FUNCTION_BLOCK Sensor_Sense
VAR_INPUT
	mxEnable: BOOL;
END_VAR
VAR_OUTPUT
	Product:STRING;
	mxINVALIDPRODUCT:BOOL;
	mxREDPLATE:BOOL;
	mxYELLOWPLATE:BOOL;
	mxBLUEPLATE:BOOL;
	mxREDCYLINDER:BOOL;
	mxYELLOWCYLINDER:BOOL;
	mxBLUECYLINDER:BOOL;
	mxREDOCTAGON:BOOL;
	mxYELLOWOCTAGON:BOOL;
	mxBLUEOCTAGON:BOOL;
	mxREDCONTAINER:BOOL;
	mxYELLOWCONTAINER:BOOL;
	mxBLUECONTAINER:BOOL;
END_VAR
VAR
	Sensor_Sense:BYTE;
END_VAR

IF mxEnable THEN
	Sensor_Sense.1:=gvl.ixInductiveSensor1;
	Sensor_Sense.2:=gvl.ixInductiveSensor2;
	Sensor_Sense.3:=gvl.ixInductiveSensor3;
	Sensor_Sense.4:=gvl.ixInductiveSensor4;
END_IF

IF Sensor_Sense = 0 OR Sensor_Sense = 4 OR Sensor_Sense = 2 OR Sensor_Sense = 6 THEN
 	Product:='InvalidPart';
	mxINVALIDPRODUCT:=FALSE;
END_IF

IF Sensor_Sense=16 THEN
	Product:='Blue Container';
	mxREDPLATE:=FALSE;
	mxYELLOWPLATE:=FALSE;
	mxBLUEPLATE:=FALSE;
	mxREDCYLINDER:=FALSE;
	mxYELLOWCYLINDER:=FALSE;
	mxBLUECYLINDER:=FALSE;
	mxREDOCTAGON:=FALSE;
	mxYELLOWOCTAGON:=FALSE;
	mxBLUEOCTAGON:=FALSE;
	mxREDCONTAINER:=FALSE;
	mxYELLOWCONTAINER:=FALSE;
	mxBLUECONTAINER:=TRUE;
	
END_IF

IF Sensor_Sense=8 THEN
	Product:='Yellow Container';
	mxREDPLATE:=FALSE;
	mxYELLOWPLATE:=FALSE;
	mxBLUEPLATE:=FALSE;
	mxREDCYLINDER:=FALSE;
	mxYELLOWCYLINDER:=FALSE;
	mxBLUECYLINDER:=FALSE;
	mxREDOCTAGON:=FALSE;
	mxYELLOWOCTAGON:=FALSE;
	mxBLUEOCTAGON:=FALSE;
	mxREDCONTAINER:=FALSE;
	mxYELLOWCONTAINER:=TRUE;
	mxBLUECONTAINER:=FALSE;
END_IF

IF Sensor_Sense=24 THEN
	Product:='Red Container';
	mxREDPLATE:=FALSE;
	mxYELLOWPLATE:=FALSE;
	mxBLUEPLATE:=FALSE;
	mxREDCYLINDER:=FALSE;
	mxYELLOWCYLINDER:=FALSE;
	mxBLUECYLINDER:=FALSE;
	mxREDOCTAGON:=FALSE;
	mxYELLOWOCTAGON:=FALSE;
	mxBLUEOCTAGON:=FALSE;
	mxREDCONTAINER:=TRUE;
	mxYELLOWCONTAINER:=FALSE;
	mxBLUECONTAINER:=FALSE;
END_IF

IF Sensor_Sense=20 THEN
	Product:='Blue Cylinder';
	mxREDPLATE:=FALSE;
	mxYELLOWPLATE:=FALSE;
	mxBLUEPLATE:=FALSE;
	mxREDCYLINDER:=FALSE;
	mxYELLOWCYLINDER:=FALSE;
	mxBLUECYLINDER:=TRUE;
	mxREDOCTAGON:=FALSE;
	mxYELLOWOCTAGON:=FALSE;
	mxBLUEOCTAGON:=FALSE;
	mxREDCONTAINER:=FALSE;
	mxYELLOWCONTAINER:=FALSE;
	mxBLUECONTAINER:=FALSE;
END_IF

IF Sensor_Sense=12 THEN
	Product:='Blue Octagon';
	mxREDPLATE:=FALSE;
	mxYELLOWPLATE:=FALSE;
	mxBLUEPLATE:=FALSE;
	mxREDCYLINDER:=FALSE;
	mxYELLOWCYLINDER:=FALSE;
	mxBLUECYLINDER:=FALSE;
	mxREDOCTAGON:=FALSE;
	mxYELLOWOCTAGON:=FALSE;
	mxBLUEOCTAGON:=TRUE;
	mxREDCONTAINER:=FALSE;
	mxYELLOWCONTAINER:=FALSE;
	mxBLUECONTAINER:=FALSE;
END_IF

IF Sensor_Sense=28 THEN
	Product:='Blue Plate';
	mxREDPLATE:=FALSE;
	mxYELLOWPLATE:=FALSE;
	mxBLUEPLATE:=TRUE;
	mxREDCYLINDER:=FALSE;
	mxYELLOWCYLINDER:=FALSE;
	mxBLUECYLINDER:=FALSE;
	mxREDOCTAGON:=FALSE;
	mxYELLOWOCTAGON:=FALSE;
	mxBLUEOCTAGON:=FALSE;
	mxREDCONTAINER:=FALSE;
	mxYELLOWCONTAINER:=FALSE;
	mxBLUECONTAINER:=FALSE;
END_IF

IF Sensor_Sense=18 THEN
	Product:='Yellow Cylinder';
	mxREDPLATE:=FALSE;
	mxYELLOWPLATE:=FALSE;
	mxBLUEPLATE:=FALSE;
	mxREDCYLINDER:=FALSE;
	mxYELLOWCYLINDER:=TRUE;
	mxBLUECYLINDER:=FALSE;
	mxREDOCTAGON:=FALSE;
	mxYELLOWOCTAGON:=FALSE;
	mxBLUEOCTAGON:=FALSE;
	mxREDCONTAINER:=FALSE;
	mxYELLOWCONTAINER:=FALSE;
	mxBLUECONTAINER:=FALSE;
END_IF

IF Sensor_Sense=10 THEN
	Product:='Yellow Octagon';
	mxREDPLATE:=FALSE;
	mxYELLOWPLATE:=FALSE;
	mxBLUEPLATE:=FALSE;
	mxREDCYLINDER:=FALSE;
	mxYELLOWCYLINDER:=FALSE;
	mxBLUECYLINDER:=FALSE;
	mxREDOCTAGON:=FALSE;
	mxYELLOWOCTAGON:=TRUE;
	mxBLUEOCTAGON:=FALSE;
	mxREDCONTAINER:=FALSE;
	mxYELLOWCONTAINER:=FALSE;
	mxBLUECONTAINER:=FALSE;
END_IF

IF Sensor_Sense=26 THEN
	Product:='Yellow Plate';
	mxREDPLATE:=FALSE;
	mxYELLOWPLATE:=TRUE;
	mxBLUEPLATE:=FALSE;
	mxREDCYLINDER:=FALSE;
	mxYELLOWCYLINDER:=FALSE;
	mxBLUECYLINDER:=FALSE;
	mxREDOCTAGON:=FALSE;
	mxYELLOWOCTAGON:=FALSE;
	mxBLUEOCTAGON:=FALSE;
	mxREDCONTAINER:=FALSE;
	mxYELLOWCONTAINER:=FALSE;
	mxBLUECONTAINER:=FALSE;
END_IF

IF Sensor_Sense=22 THEN
	Product:='Red Cylinder';
	mxREDPLATE:=FALSE;
	mxYELLOWPLATE:=FALSE;
	mxBLUEPLATE:=FALSE;
	mxREDCYLINDER:=TRUE;
	mxYELLOWCYLINDER:=FALSE;
	mxBLUECYLINDER:=FALSE;
	mxREDOCTAGON:=FALSE;
	mxYELLOWOCTAGON:=FALSE;
	mxBLUEOCTAGON:=FALSE;
	mxREDCONTAINER:=FALSE;
	mxYELLOWCONTAINER:=FALSE;
	mxBLUECONTAINER:=FALSE;
END_IF

IF Sensor_Sense=14 THEN
	Product:='Red Octagon';
	mxREDPLATE:=FALSE;
	mxYELLOWPLATE:=FALSE;
	mxBLUEPLATE:=FALSE;
	mxREDCYLINDER:=FALSE;
	mxYELLOWCYLINDER:=FALSE;
	mxBLUECYLINDER:=FALSE;
	mxREDOCTAGON:=TRUE;
	mxYELLOWOCTAGON:=FALSE;
	mxBLUEOCTAGON:=FALSE;
	mxREDCONTAINER:=FALSE;
	mxYELLOWCONTAINER:=FALSE;
	mxBLUECONTAINER:=FALSE;
END_IF

IF Sensor_Sense=30 THEN
	Product:='Red Plate';
	mxREDPLATE:=TRUE;
	mxYELLOWPLATE:=FALSE;
	mxBLUEPLATE:=FALSE;
	mxREDCYLINDER:=FALSE;
	mxYELLOWCYLINDER:=FALSE;
	mxBLUECYLINDER:=FALSE;
	mxREDOCTAGON:=FALSE;
	mxYELLOWOCTAGON:=FALSE;
	mxBLUEOCTAGON:=FALSE;
	mxREDCONTAINER:=FALSE;
	mxYELLOWCONTAINER:=FALSE;
	mxBLUECONTAINER:=FALSE;
END_IF

END_FUNCTION_BLOCK

(* stored: Version 1.1.0.1, ProductVersion 3.1.4024.12
   POU Sensor_Sense: Id {fa389c25-a045-4d57-ab3e-15214645fa9f}, SpecialFunc None *)
